# B&R Automation Studio project BenchEDM_AS6 (part 9)

#### Services_DirMan.st
```iecst
ACTION Services_DirMan:
	gVis.Services.DirMan.DirectoriesCreated										:= gMain.Services.DirMan.Out.DirectoriesCreated;
	gVis.Services.DirMan.Updating												:= gMain.Services.DirMan.Internal.CTON_Delay.IN = FALSE;
	IF NOT gVis.Services.DirMan.Updating THEN
		IF NOT gVis.Services.DirMan.UpdatingEdge THEN
			FOR Idx_FileList := 0 TO MAX_DIR_MAN_FILE_LIST_IDX DO
				gVis.Services.DirMan.FileList.Num[Idx_FileList]					:= INT_TO_UDINT(Idx_FileList);
				ascDT(UDINT_TO_DT(gMain.Services.DirMan.Out.FileList[Idx_FileList].DateUDINT), ADR(gVis.Services.DirMan.FileList.DateString[Idx_FileList]), SIZEOF(gVis.Services.DirMan.FileList.DateString[Idx_FileList]));
				gVis.Services.DirMan.FileList.Path[Idx_FileList]				:= gMain.Services.DirMan.Out.FileList[Idx_FileList].Path;
				IF Idx_FileList = 0 THEN
					gVis.Services.DirMan.FileList.Path[Idx_FileList]			:= '<ROOT>';
					gVis.Services.DirMan.FileList.DateString[Idx_FileList]		:= '-';
				END_IF;
				gVis.Services.DirMan.FileList.IsDir[Idx_FileList]				:= gMain.Services.DirMan.Out.FileList[Idx_FileList].IsDir;
				gVis.Services.DirMan.FileList.Size[Idx_FileList]				:= gMain.Services.DirMan.Out.FileList[Idx_FileList].Size;

				gVis.Services.DirMan.FileListUSB.Num[Idx_FileList]				:= INT_TO_UDINT(Idx_FileList);
				ascDT(UDINT_TO_DT(gMain.Services.DirMan.Out.FileListUSB[Idx_FileList].DateUDINT), ADR(gVis.Services.DirMan.FileListUSB.DateString[Idx_FileList]), SIZEOF(gVis.Services.DirMan.FileListUSB.DateString[Idx_FileList]));
				gVis.Services.DirMan.FileListUSB.Path[Idx_FileList]				:= gMain.Services.DirMan.Out.FileListUSB[Idx_FileList].Path;
				IF Idx_FileList = 0 AND gMain.Services.DirMan.Internal.TC_Dir_USB_Connect_0.connected THEN
					gVis.Services.DirMan.FileListUSB.Path[Idx_FileList]			:= '<ROOT>';
					gVis.Services.DirMan.FileListUSB.DateString[Idx_FileList]	:= '-';
				END_IF;
				gVis.Services.DirMan.FileListUSB.IsDir[Idx_FileList]			:= gMain.Services.DirMan.Out.FileListUSB[Idx_FileList].IsDir;
				gVis.Services.DirMan.FileListUSB.Size[Idx_FileList]				:= gMain.Services.DirMan.Out.FileListUSB[Idx_FileList].Size;
			END_FOR;
			brsmemset(ADR(gVis.Services.DirMan.TableConfig_USB),0,SIZEOF(gVis.Services.DirMan.TableConfig_USB));
			TC_brsstrcat(ADR(gVis.Services.DirMan.TableConfig_USB),ADR('{"specRows": [ {"from":'),SIZEOF(gVis.Services.DirMan.TableConfig_USB));
			gVis.Services.DirMan.TempINT										:= 0;
			FOR Idx_FileList := 0 TO MAX_DIR_MAN_FILE_LIST_IDX DO
				IF gMain.Services.DirMan.Out.FileListUSB[Idx_FileList].DateUDINT = 0 AND gMain.Services.DirMan.Out.FileListUSB[Idx_FileList].IsDir = FALSE THEN
					gVis.Services.DirMan.TempINT								:= Idx_FileList;
					EXIT;
				END_IF;
			END_FOR;
			gVis.Services.DirMan.TempSTRING 									:= INT_TO_STRING(gVis.Services.DirMan.TempINT);
			TC_brsstrcat(ADR(gVis.Services.DirMan.TableConfig_USB),ADR(gVis.Services.DirMan.TempSTRING),SIZEOF(gVis.Services.DirMan.TableConfig_USB));
			TC_brsstrcat(ADR(gVis.Services.DirMan.TableConfig_USB),ADR(', "to":'),SIZEOF(gVis.Services.DirMan.TableConfig_USB));
			gVis.Services.DirMan.TempINT										:= MAX_DIR_MAN_FILE_LIST_IDX;
			gVis.Services.DirMan.TempSTRING 									:= INT_TO_STRING(gVis.Services.DirMan.TempINT);
			TC_brsstrcat(ADR(gVis.Services.DirMan.TableConfig_USB),ADR(gVis.Services.DirMan.TempSTRING),SIZEOF(gVis.Services.DirMan.TableConfig_USB));
			TC_brsstrcat(ADR(gVis.Services.DirMan.TableConfig_USB),ADR(', "visible":false} ]}'),SIZEOF(gVis.Services.DirMan.TableConfig_USB));

			brsmemset(ADR(gVis.Services.DirMan.TableConfig_User),0,SIZEOF(gVis.Services.DirMan.TableConfig_User));
			TC_brsstrcat(ADR(gVis.Services.DirMan.TableConfig_User),ADR('{"specRows": [ {"from":'),SIZEOF(gVis.Services.DirMan.TableConfig_User));
			gVis.Services.DirMan.TempINT										:= 0;
			FOR Idx_FileList := 0 TO MAX_DIR_MAN_FILE_LIST_IDX DO
				IF gMain.Services.DirMan.Out.FileList[Idx_FileList].DateUDINT = 0 AND gMain.Services.DirMan.Out.FileList[Idx_FileList].IsDir = FALSE THEN
					gVis.Services.DirMan.TempINT								:= Idx_FileList;
					EXIT;
				END_IF;
			END_FOR;
			gVis.Services.DirMan.TempSTRING 									:= INT_TO_STRING(gVis.Services.DirMan.TempINT);
			TC_brsstrcat(ADR(gVis.Services.DirMan.TableConfig_User),ADR(gVis.Services.DirMan.TempSTRING),SIZEOF(gVis.Services.DirMan.TableConfig_User));
			TC_brsstrcat(ADR(gVis.Services.DirMan.TableConfig_User),ADR(', "to":'),SIZEOF(gVis.Services.DirMan.TableConfig_User));
			gVis.Services.DirMan.TempINT										:= MAX_DIR_MAN_FILE_LIST_IDX;
			gVis.Services.DirMan.TempSTRING 									:= INT_TO_STRING(gVis.Services.DirMan.TempINT);
			TC_brsstrcat(ADR(gVis.Services.DirMan.TableConfig_User),ADR(gVis.Services.DirMan.TempSTRING),SIZEOF(gVis.Services.DirMan.TableConfig_User));
			TC_brsstrcat(ADR(gVis.Services.DirMan.TableConfig_User),ADR(', "visible":false} ]}'),SIZEOF(gVis.Services.DirMan.TableConfig_User));
		END_IF;
		gVis.Services.DirMan.UpdatingEdge										:= TRUE;
	ELSE
		gVis.Services.DirMan.UpdatingEdge										:= FALSE;
	END_IF;
	IF gVis.Services.DirMan.SelectedIndexUSB >= 0 AND gVis.Services.DirMan.SelectedIndexUSB <= MAX_DIR_MAN_FILE_LIST_IDX THEN
		gVis.Services.DirMan.Cmd.PathUSB										:= gVis.Services.DirMan.FileListUSB.Path[gVis.Services.DirMan.SelectedIndexUSB];
		IF gVis.Services.DirMan.SelectedIndexUSB = 0 THEN
			gVis.Services.DirMan.Cmd.PathUSB									:= '/';
		END_IF;
		gVis.Services.DirMan.Cmd.DirUSB											:= gVis.Services.DirMan.FileListUSB.IsDir[gVis.Services.DirMan.SelectedIndexUSB];
	END_IF;
	IF gVis.Services.DirMan.SelectedIndexUser >= 0 AND gVis.Services.DirMan.SelectedIndexUser <= MAX_DIR_MAN_FILE_LIST_IDX THEN
		gVis.Services.DirMan.Cmd.PathUser										:= gVis.Services.DirMan.FileList.Path[gVis.Services.DirMan.SelectedIndexUser];
		IF gVis.Services.DirMan.SelectedIndexUser = 0 THEN
			gVis.Services.DirMan.Cmd.PathUser									:= '/';
		END_IF;
		gVis.Services.DirMan.Cmd.DirUser										:= gVis.Services.DirMan.FileList.IsDir[gVis.Services.DirMan.SelectedIndexUser];
	END_IF;
	gVis.Services.DirMan.USBConnected											:= gMain.Services.DirMan.Internal.TC_Dir_USB_Connect_0.connected;
	gVis.Services.DirMan.Enable_Command											:= (gVis.Services.DirMan.Cmd.Action = DIR_MAN_ACTION_COPY_TO_USB     AND gVis.Services.DirMan.Cmd.DirUSB   AND gVis.Services.DirMan.USBConnected AND NOT gVis.Services.DirMan.CmdActive)
																				OR (gVis.Services.DirMan.Cmd.Action = DIR_MAN_ACTION_COPY_TO_USER    AND gVis.Services.DirMan.Cmd.DirUser  AND gVis.Services.DirMan.USBConnected AND NOT gVis.Services.DirMan.CmdActive)
																				OR (gVis.Services.DirMan.Cmd.Action = DIR_MAN_ACTION_CREATE_DIR_USB  AND gVis.Services.DirMan.Cmd.DirUSB   AND gVis.Services.DirMan.Cmd.ParString <> '' AND gVis.Services.DirMan.USBConnected AND NOT gVis.Services.DirMan.CmdActive)
																				OR (gVis.Services.DirMan.Cmd.Action = DIR_MAN_ACTION_CREATE_DIR_USER AND gVis.Services.DirMan.Cmd.DirUser  AND gVis.Services.DirMan.Cmd.ParString <> '' AND NOT gVis.Services.DirMan.CmdActive)
																				OR (gVis.Services.DirMan.Cmd.Action = DIR_MAN_ACTION_DELETE_USB      AND gVis.Services.DirMan.USBConnected AND NOT gVis.Services.DirMan.CmdActive)
																				OR (gVis.Services.DirMan.Cmd.Action = DIR_MAN_ACTION_DELETE_USER     AND NOT gVis.Services.DirMan.CmdActive)
																				;
	IF gVis.Services.DirMan.Command THEN
		gVis.Services.DirMan.Command											:= FALSE;
		gVis.Services.DirMan.CmdActive											:= TRUE;
		gVis.Services.DirMan.ActiveCmd											:= gVis.Services.DirMan.Cmd;
	END_IF;
	IF gVis.Services.DirMan.Refresh THEN
		gVis.Services.DirMan.Refresh											:= FALSE;
		gMain.Services.DirMan.In.Refresh										:= TRUE;
	END_IF;
	IF gVis.Services.DirMan.Confirm THEN
		gVis.Services.DirMan.Confirm											:= FALSE;
		gVis.Services.DirMan.CmdActive											:= FALSE;
		IF gMain.Services.DirMan.In.TransferList[0].Valid THEN
			brsmemmove(ADR(gMain.Services.DirMan.In.TransferList)+SIZEOF(gMain.Services.DirMan.In.TransferList[0]),ADR(gMain.Services.DirMan.In.TransferList),SIZEOF(gMain.Services.DirMan.In.TransferList)-SIZEOF(gMain.Services.DirMan.In.TransferList[0]));
			brsmemset(ADR(gMain.Services.DirMan.In.TransferList[0]),0,SIZEOF(gMain.Services.DirMan.In.TransferList[0]));
		END_IF;
		CASE gVis.Services.DirMan.ActiveCmd.Action OF
			DIR_MAN_ACTION_COPY_TO_USER:
				gMain.Services.DirMan.In.TransferList[0].Valid					:= TRUE;
				gMain.Services.DirMan.In.TransferList[0].SrcOrDestUSB			:= TRUE;
				gMain.Services.DirMan.In.TransferList[0].IsDir					:= gVis.Services.DirMan.ActiveCmd.DirUSB;
				gMain.Services.DirMan.In.TransferList[0].SrcDev					:= 'USB_DEVICE';
				gMain.Services.DirMan.In.TransferList[0].SrcPath				:= gVis.Services.DirMan.ActiveCmd.PathUSB;
				gMain.Services.DirMan.In.TransferList[0].DestDev				:= gMain.Services.DeviceName;
				gMain.Services.DirMan.In.TransferList[0].DestPath				:= gVis.Services.DirMan.ActiveCmd.PathUser;
			DIR_MAN_ACTION_COPY_TO_USB:
				gMain.Services.DirMan.In.TransferList[0].Valid					:= TRUE;
				gMain.Services.DirMan.In.TransferList[0].SrcOrDestUSB			:= TRUE;
				gMain.Services.DirMan.In.TransferList[0].IsDir					:= gVis.Services.DirMan.ActiveCmd.DirUser;
				gMain.Services.DirMan.In.TransferList[0].SrcDev					:= gMain.Services.DeviceName;
				gMain.Services.DirMan.In.TransferList[0].SrcPath				:= gVis.Services.DirMan.ActiveCmd.PathUser;
				gMain.Services.DirMan.In.TransferList[0].DestDev				:= 'USB_DEVICE';
				gMain.Services.DirMan.In.TransferList[0].DestPath				:= gVis.Services.DirMan.ActiveCmd.PathUSB;
			DIR_MAN_ACTION_DELETE_USER:
				gMain.Services.DirMan.In.TransferList[0].Valid					:= TRUE;
				gMain.Services.DirMan.In.TransferList[0].NoTransfer				:= TRUE;
				gMain.Services.DirMan.In.TransferList[0].SrcDelete				:= TRUE;
				gMain.Services.DirMan.In.TransferList[0].IsDir					:= gVis.Services.DirMan.ActiveCmd.DirUser;
				gMain.Services.DirMan.In.TransferList[0].SrcDev					:= gMain.Services.DeviceName;
				gMain.Services.DirMan.In.TransferList[0].SrcPath				:= gVis.Services.DirMan.ActiveCmd.PathUser;
				gMain.Services.DirMan.In.TransferList[0].DestDev				:= gMain.Services.DeviceName;
				gMain.Services.DirMan.In.TransferList[0].DestPath				:= gVis.Services.DirMan.ActiveCmd.PathUser;
			DIR_MAN_ACTION_DELETE_USB:
				gMain.Services.DirMan.In.TransferList[0].Valid					:= TRUE;
				gMain.Services.DirMan.In.TransferList[0].NoTransfer				:= TRUE;
				gMain.Services.DirMan.In.TransferList[0].SrcDelete				:= TRUE;
				gMain.Services.DirMan.In.TransferList[0].SrcOrDestUSB			:= TRUE;
				gMain.Services.DirMan.In.TransferList[0].IsDir					:= gVis.Services.DirMan.ActiveCmd.DirUSB;
				gMain.Services.DirMan.In.TransferList[0].SrcDev					:= 'USB_DEVICE';
				gMain.Services.DirMan.In.TransferList[0].SrcPath				:= gVis.Services.DirMan.ActiveCmd.PathUSB;
				gMain.Services.DirMan.In.TransferList[0].DestDev				:= 'USB_DEVICE';
				gMain.Services.DirMan.In.TransferList[0].DestPath				:= gVis.Services.DirMan.ActiveCmd.PathUSB;
			DIR_MAN_ACTION_CREATE_DIR_USER:
				gMain.Services.DirMan.In.TransferList[0].Valid					:= TRUE;
				gMain.Services.DirMan.In.TransferList[0].NoTransfer				:= TRUE;
				gMain.Services.DirMan.In.TransferList[0].SrcCreateDir			:= TRUE;
				gMain.Services.DirMan.In.TransferList[0].IsDir					:= gVis.Services.DirMan.ActiveCmd.DirUser;
				gMain.Services.DirMan.In.TransferList[0].SrcDev					:= gMain.Services.DeviceName;
				gMain.Services.DirMan.In.TransferList[0].SrcPath				:= gVis.Services.DirMan.ActiveCmd.PathUser;
				IF gMain.Services.DirMan.In.TransferList[0].SrcPath <> '/' THEN
					TC_brsstrcat(ADR(gMain.Services.DirMan.In.TransferList[0].SrcPath),ADR('/'),SIZEOF(gMain.Services.DirMan.In.TransferList[0].SrcPath));
				END_IF;
				TC_brsstrcat(ADR(gMain.Services.DirMan.In.TransferList[0].SrcPath),ADR(gVis.Services.DirMan.ActiveCmd.ParString),SIZEOF(gMain.Services.DirMan.In.TransferList[0].SrcPath));
				gMain.Services.DirMan.In.TransferList[0].DestDev				:= gMain.Services.DeviceName;
				gMain.Services.DirMan.In.TransferList[0].DestPath				:= gVis.Services.DirMan.ActiveCmd.PathUser;
				IF gMain.Services.DirMan.In.TransferList[0].DestPath <> '/' THEN
					TC_brsstrcat(ADR(gMain.Services.DirMan.In.TransferList[0].DestPath),ADR('/'),SIZEOF(gMain.Services.DirMan.In.TransferList[0].DestPath));
				END_IF;
				TC_brsstrcat(ADR(gMain.Services.DirMan.In.TransferList[0].DestPath),ADR(gVis.Services.DirMan.ActiveCmd.ParString),SIZEOF(gMain.Services.DirMan.In.TransferList[0].DestPath));
			DIR_MAN_ACTION_CREATE_DIR_USB:
				gMain.Services.DirMan.In.TransferList[0].Valid					:= TRUE;
				gMain.Services.DirMan.In.TransferList[0].NoTransfer				:= TRUE;
				gMain.Services.DirMan.In.TransferList[0].SrcCreateDir			:= TRUE;
				gMain.Services.DirMan.In.TransferList[0].SrcOrDestUSB			:= TRUE;
				gMain.Services.DirMan.In.TransferList[0].IsDir					:= gVis.Services.DirMan.ActiveCmd.DirUSB;
				gMain.Services.DirMan.In.TransferList[0].SrcDev					:= 'USB_DEVICE';
				gMain.Services.DirMan.In.TransferList[0].SrcPath				:= gVis.Services.DirMan.ActiveCmd.PathUSB;
				IF gMain.Services.DirMan.In.TransferList[0].SrcPath <> '/' THEN
					TC_brsstrcat(ADR(gMain.Services.DirMan.In.TransferList[0].SrcPath),ADR('/'),SIZEOF(gMain.Services.DirMan.In.TransferList[0].SrcPath));
				END_IF;
				TC_brsstrcat(ADR(gMain.Services.DirMan.In.TransferList[0].SrcPath),ADR(gVis.Services.DirMan.ActiveCmd.ParString),SIZEOF(gMain.Services.DirMan.In.TransferList[0].SrcPath));
				gMain.Services.DirMan.In.TransferList[0].DestDev				:= 'USB_DEVICE';
				gMain.Services.DirMan.In.TransferList[0].DestPath				:= gVis.Services.DirMan.ActiveCmd.PathUSB;
				IF gMain.Services.DirMan.In.TransferList[0].DestPath <> '/' THEN
					TC_brsstrcat(ADR(gMain.Services.DirMan.In.TransferList[0].DestPath),ADR('/'),SIZEOF(gMain.Services.DirMan.In.TransferList[0].DestPath));
				END_IF;
				TC_brsstrcat(ADR(gMain.Services.DirMan.In.TransferList[0].DestPath),ADR(gVis.Services.DirMan.ActiveCmd.ParString),SIZEOF(gMain.Services.DirMan.In.TransferList[0].DestPath));
		END_CASE;
		brsmemset(ADR(gVis.Services.DirMan.ActiveCmd),0,SIZEOF(gVis.Services.DirMan.ActiveCmd));
		gMain.Services.DirMan.In.Refresh										:= TRUE;
	END_IF;
	IF gVis.Services.DirMan.Cancel OR brsmemcmp(ADR(gVis.Services.DirMan.ActiveCmd),ADR(gVis.Services.DirMan.Cmd),SIZEOF(gVis.Services.DirMan.Cmd)) <> 0 THEN
		gVis.Services.DirMan.Cancel												:= FALSE;
		gVis.Services.DirMan.CmdActive											:= FALSE;
		brsmemset(ADR(gVis.Services.DirMan.ActiveCmd),0,SIZEOF(gVis.Services.DirMan.ActiveCmd));
	END_IF;
	gVis.Services.DirMan.CmdInactive											:= NOT gVis.Services.DirMan.CmdActive;
	gVis.Services.DirMan.Busy													:= gMain.Services.DirMan.Internal.State <> DIR_MAN_DELAY;
END_ACTION
```

#### Settings.st
```iecst
ACTION Settings:

	gVis.Settings.Save.Modified												:= FALSE;
	IF brsmemcmp(ADR(gVis.Settings.ParCmp),ADR(gVis.Settings.Par),SIZEOF(gPar)) <> 0 THEN
		gVis.Settings.Save.Modified											:= TRUE;
		IF gVis.Settings.Save.Save THEN
			gPar 															:= gVis.Settings.Par;
			gVis.Settings.ParCmp 											:= gPar;
		ELSIF gVis.Settings.Save.Cancel THEN
			gVis.Settings.Par 												:= gPar;
			gVis.Settings.ParCmp 											:= gPar;
		END_IF;
	END_IF;
	gVis.Settings.Save.Save 												:= FALSE;
	gVis.Settings.Save.Cancel 												:= FALSE;
	IF brsmemcmp(ADR(gVis.Settings.ParCmp),ADR(gPar),SIZEOF(gPar)) <> 0 THEN
		// Vis structures needs to be updated from gPar because gPar changed
		gVis.Settings.Par 													:= gPar;
		gVis.Settings.ParCmp 												:= gPar;
	END_IF;

END_ACTION
```

#### Alarms_Active.st
```iecst
ACTION Alarms_Active:

	gVis.Alarms.Active.UIConnect.AlarmList.SelectedIndex					:= gVis.Alarms.Active.SelectedIndex;
	IF gVis.Alarms.Active.Reset THEN
		gVis.Alarms.Active.Reset											:= FALSE;
		gMain.ErrorReset													:= TRUE;
	END_IF;
	gVis.Alarms.Active.UIConnect.AlarmList.PageUp							:= gVis.Alarms.Active.PageUp;
	gVis.Alarms.Active.PageUp												:= FALSE;
	gVis.Alarms.Active.UIConnect.AlarmList.PageDown							:= gVis.Alarms.Active.PageDown;
	gVis.Alarms.Active.PageDown												:= FALSE;

	brsmemset(ADR(gVis.Alarms.Active.TableConfig),0,SIZEOF(gVis.Alarms.Active.TableConfig));
	TC_brsstrcat(ADR(gVis.Alarms.Active.TableConfig),ADR('{"specRows": [ {"from":'),SIZEOF(gVis.Alarms.Active.TableConfig));
	IF gVis.Alarms.Active.UIConnect.AlarmList.MaxSelection = 0 THEN
		IF gVis.Alarms.Active.UIConnect.AlarmList.Timestamp[0] = '' THEN
			gVis.Alarms.Active.TempINT										:= 0;
		ELSE
			gVis.Alarms.Active.TempINT										:= 1;
		END_IF;
	ELSE
		gVis.Alarms.Active.TempINT											:= UINT_TO_INT(gVis.Alarms.Active.UIConnect.AlarmList.MaxSelection)+1;
	END_IF;
	gVis.Alarms.Active.TempSTRING 											:= INT_TO_STRING(gVis.Alarms.Active.TempINT);
	TC_brsstrcat(ADR(gVis.Alarms.Active.TableConfig),ADR(gVis.Alarms.Active.TempSTRING),SIZEOF(gVis.Alarms.Active.TableConfig));
	TC_brsstrcat(ADR(gVis.Alarms.Active.TableConfig),ADR(', "to":'),SIZEOF(gVis.Alarms.Active.TableConfig));
	gVis.Alarms.Active.TempINT												:= 49;
	gVis.Alarms.Active.TempSTRING 											:= INT_TO_STRING(gVis.Alarms.Active.TempINT);
	TC_brsstrcat(ADR(gVis.Alarms.Active.TableConfig),ADR(gVis.Alarms.Active.TempSTRING),SIZEOF(gVis.Alarms.Active.TableConfig));
	TC_brsstrcat(ADR(gVis.Alarms.Active.TableConfig),ADR(', "visible":false} ]}'),SIZEOF(gVis.Alarms.Active.TableConfig));

END_ACTION
```

#### Alarms_History.st
```iecst
ACTION Alarms_History:

	gVis.Alarms.History.UIConnect.AlarmList.SelectedIndex					:= gVis.Alarms.History.SelectedIndex;
	gVis.Alarms.History.UIConnect.AlarmList.PageUp							:= gVis.Alarms.History.PageUp;
	gVis.Alarms.History.PageUp												:= FALSE;
	gVis.Alarms.History.UIConnect.AlarmList.PageDown						:= gVis.Alarms.History.PageDown;
	gVis.Alarms.History.PageDown											:= FALSE;
	gMain.Services.Alarms.In.ClearHistory									:= gVis.Alarms.History.Clear;
	gVis.Alarms.History.Clear												:= FALSE;
	gMain.Services.Alarms.In.ExportHistory									:= gVis.Alarms.History.Export;
	gVis.Alarms.History.Export												:= FALSE;
	// Below loop sets the state variable to 1. Non 1 values are filtered from the table. This filters the history to only have when the alarm was triggered and not when it was acknowledged.
	FOR Idx_AlarmList := 0 TO 49 DO
		gVis.Alarms.History.State[Idx_AlarmList] 										:= 0;
		IF gVis.Alarms.History.UIConnect.AlarmList.NewState[Idx_AlarmList] = mpALARMX_STATE_ACTIVE THEN
			gVis.Alarms.History.State[Idx_AlarmList] 									:= 1;
		END_IF;
	END_FOR;

	brsmemset(ADR(gVis.Alarms.History.TableConfig),0,SIZEOF(gVis.Alarms.History.TableConfig));
	TC_brsstrcat(ADR(gVis.Alarms.History.TableConfig),ADR('{"specRows": [ {"from":'),SIZEOF(gVis.Alarms.History.TableConfig));
	IF gVis.Alarms.History.UIConnect.AlarmList.MaxSelection = 0 THEN
		IF gVis.Alarms.History.UIConnect.AlarmList.Timestamp[0] = '' THEN
			gVis.Alarms.History.TempINT										:= 0;
		ELSE
			gVis.Alarms.History.TempINT										:= 1;
		END_IF;
	ELSE
		gVis.Alarms.History.TempINT											:= UINT_TO_INT(gVis.Alarms.History.UIConnect.AlarmList.MaxSelection)+1;
	END_IF;
	gVis.Alarms.History.TempSTRING 											:= INT_TO_STRING(gVis.Alarms.History.TempINT);
	TC_brsstrcat(ADR(gVis.Alarms.History.TableConfig),ADR(gVis.Alarms.History.TempSTRING),SIZEOF(gVis.Alarms.History.TableConfig));
	TC_brsstrcat(ADR(gVis.Alarms.History.TableConfig),ADR(', "to":'),SIZEOF(gVis.Alarms.History.TableConfig));
	gVis.Alarms.History.TempINT												:= 49;
	gVis.Alarms.History.TempSTRING 											:= INT_TO_STRING(gVis.Alarms.History.TempINT);
	TC_brsstrcat(ADR(gVis.Alarms.History.TableConfig),ADR(gVis.Alarms.History.TempSTRING),SIZEOF(gVis.Alarms.History.TableConfig));
	TC_brsstrcat(ADR(gVis.Alarms.History.TableConfig),ADR(', "visible":false} ]}'),SIZEOF(gVis.Alarms.History.TableConfig));

END_ACTION
```

### Program Logical/StepDir (ReAction)

#### Variables.var
```iecst
VAR
	rtiDout_Direction : rtiDout;
	rtiDout_Step : rtiDout;
	rtiComp_0 : rtiComp;
	rtiPar_Set : rtiPar;
	rtiPar_Home : rtiPar;
	rtiRes_Act : rtiRes;
	rtiVarRead_0 : rtiVarRead;
	rtiVarWrite_0 : rtiVarWrite;
	rtiSub_0 : rtiSub;
	rtiComp_1 : rtiComp;
	rtiAdd_0 : rtiAdd;
	rtiAnd_0 : rtiAnd;
	rtiMux_1 : rtiMux;
	rtiMux_0 : rtiMux;
	rtiVarRead_1 : rtiVarRead;
	rtiVarWrite_1 : rtiVarWrite;
	rtiAdd_1 : rtiAdd;
	rtiMul_0 : rtiMul;
	rtiTP_0 : rtiTP;
	rtiDelay_0 : rtiDelay;
	rtiXor_0 : rtiXor;
	rtiNot_0 : rtiNot;
	rtiComp_2 : rtiComp;
	rtiSRff_0 : rtiSRff;
	rtiPar_DelayCount : rtiPar;
	rtiCount_0 : rtiCount;
	rtiVarRead_2 : rtiVarRead;
	rtiVarWrite_2 : rtiVarWrite;
	rtiComp_3 : rtiComp;
END_VAR
```

- Cyclic.rti (not shown)

### Program Logical/Dev (IEC)

#### Variables.var
```iecst
VAR
	MpAxisBasic_R_Y : MpAxisBasic;
	MpAxisBasicPar_R_Y : MpAxisBasicParType;
	MpAxisBasic_R_X : MpAxisBasic;
	MpAxisBasicPar_R_X : MpAxisBasicParType;
	MpAxisBasic_R_V : MpAxisBasic;
	MpAxisBasicPar_R_V : MpAxisBasicParType;
	MpAxisBasic_R_T : MpAxisBasic;
	MpAxisBasicPar_R_T : MpAxisBasicParType;
	MC_BR_TorqueControl_R_T : MC_BR_TorqueControl;
	EnableTorqueControl : BOOL;
	TC_FrSky_USB_0 : TC_FrSky_USB;
	FRM_xopen_0 : FRM_xopen;
	test : BOOL;
	UdpOpen_0 : UdpOpen;
	UdpRecv_0 : UdpRecv;
	Data : STRING[100];
END_VAR
```

#### Main.st
```iecst
PROGRAM _INIT

//	MC_BR_TorqueControl_R_T.Torque 				:= 0.1;
//	MC_BR_TorqueControl_R_T.TorqueRamp 			:= 0.01;
//	MC_BR_TorqueControl_R_T.Acceleration 		:= 1000000.0;
//	MC_BR_TorqueControl_R_T.MaximumVelocity 	:= 100.0;
//	MC_BR_TorqueControl_R_T.MinimumVelocity 	:= -100.0;

END_PROGRAM

PROGRAM _CYCLIC
//	IF UdpOpen_0.ident = 0 THEN
//		UdpOpen_0(enable := TRUE);
//	END_IF;
//	UdpRecv_0(enable := TRUE, ident := UdpOpen_0.ident, pData := ADR(Data), datamax := SIZEOF(Data)-1);
//
//
	TC_FrSky_USB_0();
//
//	MpAxisBasic_R_X(MpLink := ADR(gAxis_R_X), Enable := TRUE, ErrorReset := gMain.ErrorReset, Parameters := ADR(MpAxisBasicPar_R_X));
//	IF MpAxisBasic_R_X.UpdateDone THEN
//		MpAxisBasic_R_X.Update := FALSE;
//	END_IF;
//
//	MpAxisBasic_R_Y(MpLink := ADR(gAxis_R_Y), Enable := TRUE, ErrorReset := gMain.ErrorReset, Parameters := ADR(MpAxisBasicPar_R_Y));
//	IF MpAxisBasic_R_Y.UpdateDone THEN
//		MpAxisBasic_R_Y.Update := FALSE;
//	END_IF;
//
//	MpAxisBasic_R_V(MpLink := ADR(gAxis_R_V), Enable := TRUE, ErrorReset := gMain.ErrorReset, Parameters := ADR(MpAxisBasicPar_R_V));
//	IF MpAxisBasic_R_V.UpdateDone THEN
//		MpAxisBasic_R_V.Update := FALSE;
//	END_IF;
//
//	MpAxisBasic_R_T(MpLink := ADR(gAxis_R_T), Enable := TRUE, ErrorReset := gMain.ErrorReset, Parameters := ADR(MpAxisBasicPar_R_T));
//	IF MpAxisBasic_R_T.UpdateDone THEN
//		MpAxisBasic_R_T.Update := FALSE;
//	END_IF;
//
//	IF MC_BR_TorqueControl_R_T.Error THEN
//		EnableTorqueControl := FALSE;
//	END_IF;
//	IF MC_BR_TorqueControl_R_T.Ready THEN
//		IF EnableTorqueControl AND NOT MC_BR_TorqueControl_R_T.Active THEN
//			MC_BR_TorqueControl_R_T.Start := TRUE;
//		ELSIF NOT EnableTorqueControl AND MC_BR_TorqueControl_R_T.Active THEN
//			MC_BR_TorqueControl_R_T.Stop := TRUE;
//		END_IF;
//	END_IF;
//	MC_BR_TorqueControl_R_T(Axis := ADR(gAxis_R_T));
//	MC_BR_TorqueControl_R_T.Start := FALSE;
//	MC_BR_TorqueControl_R_T.Stop := FALSE;
//	IF MC_BR_TorqueControl_R_T.DataInitialized THEN
//		MC_BR_TorqueControl_R_T.InitData := FALSE;
//	END_IF;

END_PROGRAM

PROGRAM _EXIT

END_PROGRAM
```

### Program Logical/NGRC (IEC)

#### Types.typ
```iecst
TYPE
    MyApp_Theta_typ : STRUCT
	    Row : DINT;
        Col : DINT;
        M : ARRAY[0..MY_MAX_THETA_IDX] OF LREAL;
    END_STRUCT;
    MyApp_P_typ : STRUCT
        Row : DINT;
        Col : DINT;
        M : ARRAY[0..MY_MAX_P_IDX] OF LREAL;
    END_STRUCT;
    MyApp_History_typ : STRUCT
        Row : DINT;
        Col : DINT;
        M : ARRAY[0..MY_MAX_HISTORY_IDX] OF LREAL;
    END_STRUCT;
    MyApp_Features_typ : STRUCT
	    Row : DINT;
        Col : DINT;
        M : ARRAY[0..MY_MAX_FEATURES_IDX] OF LREAL;
    END_STRUCT;
    MyApp_SharedWorkspace_typ : STRUCT
        Row : DINT;
        Col : DINT;
        M : ARRAY[0..MY_MAX_SHARED_WORKSPACE_IDX] OF LREAL;
    END_STRUCT;
END_TYPE
```

#### Variables.var
```iecst
VAR
	MTBasicsTransferFcn_0 : MTBasicsTransferFcn;
	Omega : REAL := 4.0;
	Zeta : REAL := 0.1;
	Theta : ARRAY[0..MY_MAX_VARIABLES_IDX] OF MyApp_Theta_typ;
	P : ARRAY[0..MY_MAX_VARIABLES_IDX] OF MyApp_P_typ;
	History : ARRAY[0..MY_MAX_VARIABLES_IDX] OF MyApp_History_typ;
	Features : MyApp_Features_typ;
	SharedWorkspace : MyApp_SharedWorkspace_typ;
	Initialized : BOOL := FALSE;
	NumVariables : DINT;
	LagOrder : DINT;
	PolyOrder : DINT;
	UseBias : BOOL;
	Stride : DINT := 1;
	EnableWorkspaceReuse : BOOL;
	Output : TC_NGRC_CalcMem_Output_typ;
	TC_NGRC_Continuous_0 : TC_NGRC_Continuous;
END_VAR
VAR CONSTANT
	MY_MAX_VARIABLES_IDX : DINT := 1;
	MY_MAX_THETA_IDX : DINT := 65;
	MY_MAX_P_IDX : DINT := 4355;
	MY_MAX_HISTORY_IDX : DINT := 4;
	MY_MAX_FEATURES_IDX : DINT := 65;
	MY_MAX_SHARED_WORKSPACE_IDX : DINT := 65;
END_VAR
VAR
	FirstScanComplete : BOOL;
	i : DINT;
END_VAR
```

#### Main.st
```iecst
PROGRAM _INIT

	(* Configure Transfer Function *)
	Omega := 4.0;
	Zeta := 0.1;

END_PROGRAM

PROGRAM _CYCLIC

	MTBasicsTransferFcn_0.Numerator[0] := Omega * Omega;
	MTBasicsTransferFcn_0.Denominator[0] := Omega * Omega;
	MTBasicsTransferFcn_0.Denominator[1] := 2.0 * Zeta * Omega;
	MTBasicsTransferFcn_0.Denominator[2] := 1.0;
	MTBasicsTransferFcn_0(Enable := TRUE, Mode := mtBASICS_CONTINUOUS_TRANSFER_FCN);

	IF NOT FirstScanComplete AND TC_NGRC_Continuous_0.In.Cmd.Enable THEN
		(* Configure TC_NGRC_Continuous_0 *)
		TC_NGRC_Continuous_0.In.Par.NumVariables := MY_MAX_VARIABLES_IDX+1;
		TC_NGRC_Continuous_0.In.Par.LagOrder := 5;
		TC_NGRC_Continuous_0.In.Par.PolyOrder := 2;
		TC_NGRC_Continuous_0.In.Par.UseBias := TRUE;
		TC_NGRC_Continuous_0.In.Par.PredictionSteps := 5;
		TC_NGRC_Continuous_0.In.Par.Lambda := 0.999;
		TC_NGRC_Continuous_0.In.Par.InitVariance := 1000.0;
		(* Assign memory pointers *)
		TC_NGRC_Continuous_0.In.Par.pTheta := ADR(Theta);
		TC_NGRC_Continuous_0.In.Par.ThetaStride_Bytes := SIZEOF(Theta[0]);
		TC_NGRC_Continuous_0.In.Par.pP := ADR(P);
		TC_NGRC_Continuous_0.In.Par.PStride_Bytes := SIZEOF(P[0]);
		TC_NGRC_Continuous_0.In.Par.pHistory := ADR(History);
		TC_NGRC_Continuous_0.In.Par.HistoryStride_Bytes := SIZEOF(History[0]);
		TC_NGRC_Continuous_0.In.Par.pFeatures := ADR(Features);
		TC_NGRC_Continuous_0.In.Par.pSharedWorkspace := ADR(SharedWorkspace);

		(* Initialize dimensions *)
		FOR i := 0 TO MY_MAX_VARIABLES_IDX DO
			Theta[i].Row := MY_MAX_THETA_IDX+1; Theta[i].Col := 1;
			P[i].Row := MY_MAX_THETA_IDX+1; P[i].Col := MY_MAX_THETA_IDX+1;
			History[i].Row := MY_MAX_HISTORY_IDX+1; History[i].Col := 1;
		END_FOR;
		Features.Row := MY_MAX_FEATURES_IDX+1; Features.Col := 1;
		SharedWorkspace.Row := MY_MAX_SHARED_WORKSPACE_IDX+1; SharedWorkspace.Col := 1;

		TC_NGRC_Continuous_0.In.Cmd.Init := TRUE;
		FirstScanComplete := TRUE;
	END_IF;

	TC_NGRC_Continuous_0.In.Signal.NewSample[0] := (REAL_TO_LREAL(MTBasicsTransferFcn_0.Out)-TC_NGRC_Continuous_0.In.Signal.NewSample[1])/0.001;
	TC_NGRC_Continuous_0.In.Signal.NewSample[1] := REAL_TO_LREAL(MTBasicsTransferFcn_0.Out);
	TC_NGRC_Continuous_0();
	TC_NGRC_Continuous_0.In.Cmd.Init := FALSE;

	TC_NGRC_CalcMem(NumVariables,LagOrder,PolyOrder,UseBias,Stride,EnableWorkspaceReuse,ADR(Output));
END_PROGRAM

//PROGRAM MyApplication
//VAR
//	(* Optimally-sized arrays from calculator *)
//	Theta : ARRAY[0..5] OF MyApp_Theta_typ;
//	P : ARRAY[0..5] OF MyApp_P_typ;
//	History : ARRAY[0..5] OF MyApp_History_typ;
//	Features : MyApp_Features_typ;
//	SharedWorkspace : MyApp_SharedWorkspace_typ;
//
//	TC_NGRC_Continuous_0 : TC_NGRC_Continuous;
//
//	FirstScan : BOOL := TRUE;
//END_VAR
//
//IF FirstScan THEN
//
//	(* Configure TC_NGRC_Continuous_0 *)
//	TC_NGRC_Continuous_0.In.Par.NumVariables := 6;
//	TC_NGRC_Continuous_0.In.Par.LagOrder := 2;
//	TC_NGRC_Continuous_0.In.Par.PolyOrder := 1;
//	TC_NGRC_Continuous_0.In.Par.UseBias := TRUE;
//	TC_NGRC_Continuous_0.In.Par.PredictionSteps := 3;
//	TC_NGRC_Continuous_0.In.Par.Lambda := 0.999;
//	TC_NGRC_Continuous_0.In.Par.InitVariance := 1000.0;
//
//	(* Assign memory pointers *)
//	TC_NGRC_Continuous_0.In.Par.pTheta := ADR(Theta[0]);
//	TC_NGRC_Continuous_0.In.Par.pP := ADR(P[0]);
//	TC_NGRC_Continuous_0.In.Par.pHistory := ADR(History[0]);
//	TC_NGRC_Continuous_0.In.Par.pFeatures := ADR(Features);
//	TC_NGRC_Continuous_0.In.Par.pSharedWorkspace := ADR(SharedWorkspace);
//
//	(* NEW: Set stride values using SIZEOF *)
//	TC_NGRC_Continuous_0.In.Par.ThetaStride_Bytes := SIZEOF(MyApp_Theta_typ);
//	TC_NGRC_Continuous_0.In.Par.PStride_Bytes := SIZEOF(MyApp_P_typ);
//	TC_NGRC_Continuous_0.In.Par.HistoryStride_Bytes := SIZEOF(MyApp_History_typ);
//
//	(* Initialize dimensions *)
//	FOR i := 0 TO 5 DO
//		Theta[i].Row := 13; Theta[i].Col := 1;
//		P[i].Row := 13; P[i].Col := 13;
//		History[i].Row := 2; History[i].Col := 1;
//	END_FOR;
//	Features.Row := 13; Features.Col := 1;
//	SharedWorkspace.Row := 13; SharedWorkspace.Col := 1;
//
//	TC_NGRC_Continuous_0.In.Cmd.Init := TRUE;
//	FirstScan := FALSE;
//END_IF;
//
//(* Every cycle *)
//TC_NGRC_Continuous_0.In.Signal.NewSample := SensorValues;
//TC_NGRC_Continuous_0.In.Cmd.Enable := TRUE;
//TC_NGRC_Continuous_0();
//
//IF TC_NGRC_Continuous_0.Out.Status.Ready THEN
//	Predictions := TC_NGRC_Continuous_0.Out.Signal.Prediction[0, 0];
//END_IF;
//
//END_PROGRAM
```

### Variables.var
```iecst
VAR
	rtiDout_Direction : rtiDout;
	rtiDout_Step : rtiDout;
	rtiComp_0 : rtiComp;
	rtiPar_Set : rtiPar;
	rtiPar_Home : rtiPar;
	rtiRes_Act : rtiRes;
	rtiVarRead_0 : rtiVarRead;
	rtiVarWrite_0 : rtiVarWrite;
	rtiSub_0 : rtiSub;
	rtiComp_1 : rtiComp;
	rtiAdd_0 : rtiAdd;
	rtiAnd_0 : rtiAnd;
	rtiMux_1 : rtiMux;
	rtiMux_0 : rtiMux;
	rtiVarRead_1 : rtiVarRead;
	rtiVarWrite_1 : rtiVarWrite;
	rtiAdd_1 : rtiAdd;
	rtiMul_0 : rtiMul;
	rtiTP_0 : rtiTP;
	rtiDelay_0 : rtiDelay;
	rtiXor_0 : rtiXor;
	rtiNot_0 : rtiNot;
	rtiComp_2 : rtiComp;
	rtiSRff_0 : rtiSRff;
END_VAR
```

- Cyclic.rti (not shown)

Listed in the project but not available here: Logical/BuildVersion/BuildVer, Logical/BuildVersion/BuildVersion.typ, Logical/Libraries/TC_General/Constants.var, Logical/Libraries/TC_General/TC_General.fun, Logical/Libraries/TC_General/CTON.st, Logical/Libraries/TC_Version/Types.typ, Logical/Libraries/TC_Version/Constants.var, Logical/Libraries/TC_Version/TC_Version.fun, Logical/Libraries/TC_IO/Constants.var, Logical/Libraries/TC_Dir/Constants.var, Logical/Libraries/TC_Convert/Constants.var, Logical/Libraries/TC_ItemX/Constants.var, Logical/Libraries/TC_Array/Types.typ, Logical/Libraries/TC_SysErr/Constants.var, Logical/Libraries/TC_Recipe/Constants.var, Logical/Libraries/TC_Sim/Constants.var, Logical/Libraries/TC_Str/Constants.var, Logical/Libraries/TC_RAND/Types.typ, Logical/Libraries/TC_RAND/Constants.var, Logical/Libraries/TC_RAND/TC_RAND.fun, Logical/Libraries/TC_FrSky/Constants.var, Logical/Process/InputMan/Types.typ, Logical/Process/InputMan/Variables.var, Logical/Process/InputMan/InputDrivers, Logical/Process/Monitor/Types.typ, Logical/Process/Seq_MASTER/Types.typ, Logical/Process/OutputMan/Types.typ, Logical/Process/OutputMan/Variables.var, Logical/Services/Types.typ, Logical/Vis/Types.typ
